FUNCTION_BLOCK ServoNC EXTENDS FBA_Drive IMPLEMENTS I_EncodedDrive
VAR_OUTPUT	
	ready : BOOL;
	position : LREAL;
END_VAR
VAR
	axis : AXIS_REF;
	
	mcReadPosition : MC_ReadActualPosition;
	mcReset : MC_Reset;
	
	mcPower : MC_Power;
	mcMoveAbsolute : MC_MoveAbsolute;
	mcMoveRelative : MC_MoveRelative;
	mcMoveVelocity : MC_MoveVelocity;
	
	mcSetPosition : MC_SetPosition;
	mcStop : MC_Stop;
END_VAR
VAR_STAT CONSTANT
	targetingVelocity : INT := 500;
	continuousVelocity : INT := 200;
END_VAR

IF home OR outerLimit OR innerLimit THEN
	stop();
END_IF

blocks();

mcReset.Execute := FALSE;
mcMoveAbsolute.Execute := FALSE;
mcMoveRelative.Execute := FALSE;
mcMoveVelocity.Execute := FALSE;
mcSetPosition.Execute := FALSE;
mcStop.Execute := FALSE;

blocks();

ready := bEnable AND NOT busy AND homeSet;

METHOD PRIVATE blocks : BOOL
mcReadPosition(
	Axis:= axis, 
	Enable:= TRUE, 
	Valid=> , 
	Busy=> , 
	Error=> , 
	ErrorID=> , 
	Position=> position);

mcReset(
	Axis:= axis, 
	Execute:= , 
	Done=> , 
	Busy=> , 
	Error=> , 
	ErrorID=> );

mcPower(
	Axis:= axis, 
	Enable:= bEnable, 
	Enable_Positive:= TRUE, 
	Enable_Negative:= TRUE, 
	Override:= 100, 
	BufferMode:= , 
	Options:= , 
	Status=> , 
	Busy=> , 
	Active=> , 
	Error=> , 
	ErrorID=> );

mcMoveAbsolute(
	Axis:= axis, 
	Execute:= , 
	Position:= , 
	Velocity:= targetingVelocity, 
	Acceleration:= , 
	Deceleration:= , 
	Jerk:= , 
	BufferMode:= , 
	Options:= , 
	Done=> , 
	Busy=> , 
	Active=> , 
	CommandAborted=> , 
	Error=> , 
	ErrorID=> );
	
mcMoveRelative(
	Axis:= axis, 
	Execute:= , 
	Distance:= ,
	Velocity:= targetingVelocity, 
	Acceleration:= , 
	Deceleration:= , 
	Jerk:= , 
	BufferMode:= , 
	Options:= , 
	Done=> , 
	Busy=> , 
	Active=> , 
	CommandAborted=> , 
	Error=> , 
	ErrorID=> );
	
mcMoveVelocity( //stopped with stop();
	Axis:= axis, 
	Execute:= , 
	Velocity:= continuousVelocity, 
	Acceleration:= , 
	Deceleration:= , 
	Jerk:= , 
	Direction:= , 
	BufferMode:= , 
	Options:= , 
	InVelocity=> , 
	Busy=> , 
	Active=> , 
	CommandAborted=> , 
	Error=> , 
	ErrorID=> );
	
mcSetPosition(
	Axis:= axis, 
	Execute:= , 
	Position:= , 
	Mode:= , 
	Options:= , 
	Done=> , 
	Busy=> , 
	Error=> , 
	ErrorID=> );
	
mcStop(
	Axis:= axis, 
	Execute:= , 
	Deceleration:= , 
	Jerk:= , 
	Options:= , 
	Done=> , 
	Busy=> , 
	Active=> , 
	CommandAborted=> , 
	Error=> , 
	ErrorID=> );
END_METHOD

PROPERTY Busy : BOOL
GET
busy := 
	mcMoveAbsolute.Busy OR 
	mcMoveRelative.Busy OR 
	mcMoveVelocity.Busy OR 
	mcSetPosition.Busy OR 
	mcReset.Busy OR 
	mcStop.Busy OR 
	step <> 0;
END_GET
END_PROPERTY

PROPERTY CurrentPosition : LREAL
GET
CurrentPosition := position;
END_GET
SET
position := CurrentPosition;
END_SET
END_PROPERTY

PROPERTY Error : BOOL
GET
error := 
	mcMoveAbsolute.Error OR 
	mcMoveRelative.Error OR 
	mcMoveVelocity.Error OR 
	mcSetPosition.Error OR 
	mcReset.Error OR 
	mcStop.Error;
END_GET
END_PROPERTY

METHOD homingSequence : BOOL
CASE step OF
	Homing.IDLE:
		IF bEnable THEN
			step := Homing.IN;
		END_IF
		
	Homing.IN:
		IF mcMoveVelocity.Execute AND NOT innerLimit THEN
			mcMoveVelocity.Execute := FALSE;
			step := Homing.OUT;
			RETURN;
		END_IF
		
		mcMoveVelocity.Direction := MC_Negative_Direction;
		mcMoveVelocity.Execute := TRUE;
		
	Homing.OUT:
		IF mcMoveVelocity.Execute AND NOT home THEN //if reached home
			mcMoveVelocity.Execute := FALSE;
			step := Homing.STOP;
			RETURN;
		END_IF
		
		mcMoveVelocity.Direction := MC_Positive_Direction;
		mcMoveVelocity.Execute := TRUE;
		
	Homing.STOP:
		IF mcStop.Execute AND mcStop.Done THEN
			mcStop.Execute := FALSE;
			step := Homing.SET;
			RETURN;
		END_IF
		
		mcStop.Execute := TRUE;
		
	Homing.SET:
		IF mcSetPosition.Execute AND mcSetPosition.Done THEN
			mcSetPosition.Execute := FALSE;
			homingSequence := TRUE;
			step := Homing.IDLE;
			RETURN;
		END_IF
		
		mcSetPosition.Position := 0;
		mcSetPosition.Execute := TRUE;
		
END_CASE
END_METHOD

METHOD moveAbsolute : BOOL
VAR_INPUT
	newTarget : LREAL;
END_VAR
(*
VAR_OUTPUT
	fault : BOOL;
END_VAR
*)
IF NOT busy AND NOT error THEN
	mcMoveAbsolute.Position := newTarget;
	mcMoveAbsolute.Execute := TRUE;
END_IF

moveAbsolute := (*mcMoveAbsolute.Done AND mcMoveAbsolute.Active;*)
	position = newTarget;
END_METHOD

METHOD moveContinuous : BOOL
VAR_INPUT
	//direction : BOOL; //direction (F = inwards, T = outwards)
	direction : MC_Direction;
END_VAR
(*
IF mcMoveVelocity.Active THEN
	stop();
END_IF

IF NOT mcStop.Done THEN
	RETURN;
END_IF
*)
(*
IF direction THEN
	mcMoveVelocity.Direction := MC_Positive_Direction;
ELSE
	mcMoveVelocity.Direction := MC_Negative_Direction;
END_IF
*)
mcMoveVelocity.Direction := direction;

IF NOT mcMoveVelocity.Error THEN
	mcMoveVelocity.Execute := TRUE;
	moveContinuous := TRUE;
END_IF
END_METHOD

METHOD moveRelative : BOOL
VAR_INPUT
	distance : LREAL;
END_VAR
mcMoveRelative.Distance := distance;

moveRelative := mcMoveRelative.Done;
END_METHOD

METHOD reset : BOOL
VAR_INPUT
END_VAR
mcReset.Execute := TRUE;

reset := mcReset.Done;
END_METHOD

METHOD stop : BOOL
VAR_INPUT
END_VAR
mcStop.Execute := TRUE;
END_METHOD

PROPERTY TargetPosition : LREAL
GET
END_GET
SET
moveAbsolute(newTarget := TargetPosition);
END_SET
END_PROPERTY

END_FUNCTION_BLOCK

(* stored: Version 1.1.0.1, ProductVersion 3.1.4024.11
   POU ServoNC: Id {f939ae28-30bd-4997-8b95-af50702e8d64}, SpecialFunc None
   Folder Properties: Id {f4fb86df-136f-4996-9daa-b3b8a4b4fe75}
   Method blocks: Id {4f4b3711-209a-4326-9f5b-d1908f737531}
   Property Busy: Id {76e617c1-1707-418c-afd8-37e3d0a70099}
   Get Get: Id {9821e814-6021-4995-a4d6-e74adde35b23}
   Property CurrentPosition: Id {552cdbb0-b891-4b67-ad01-a8cfc1c516eb}
   Get Get: Id {f42f05dd-f56e-4930-a286-1888d4d594cd}
   Set Set: Id {cba03562-eb55-4743-94dc-7cf01962b58c}
   Property Error: Id {7daf4b31-4ccd-4ebb-b598-fd16e9795a78}
   Get Get: Id {edbd4fca-a224-4fe5-ba01-ff917580b072}
   Method homingSequence: Id {c889c79b-08e7-46ba-b03a-e3652fe9a7a9}
   Method moveAbsolute: Id {9a0c1523-e496-48d2-89d9-d71629c86307}
   Method moveContinuous: Id {c1bd97e2-f7e7-45ed-bf81-7afd3b7c53ff}
   Method moveRelative: Id {a4516e41-c115-4d38-aa54-f9462db8dc0d}
   Method reset: Id {b7706fbc-8e49-4562-bc6d-21f87f45b14e}
   Method stop: Id {131a01d5-9f85-446c-9242-ad02c99596c6}
   Property TargetPosition: Id {222c0d80-2607-4af6-8461-be098758948d}
   Get Get: Id {b917e1f8-7faf-4ca9-8c30-5bfbcfdfaf97}
   Set Set: Id {f401d7bc-6585-4a9b-ae06-cd3e51203159} *)
